_CFC_ (* Continuous Function Chart, elements in execution order *)
#0 SHU6_P2_M_MAXSPEED <= SHU6_P2_M_MAXSPEED_CH
#1 <>(SHU6_P2_M_MAXSPEED_CH, SHU6_P2_M_MAXSPEED_CH_OLD)
#2 RS_RUCH:RS(SET: #1, RESET1: #4.Q)
#3 V_RUCH <= #2.Q1
#4 TON_RUCH:TON(IN: #2.Q1, PT: T#10s)
#5 AND(SHU6_P2_YA3_M_UST_VKL_UVEL_CHAST, SHU6_P2_YA4_M_UST_VKL_UVEL_CHAST, SHU6_P2_UST_RE_RABOTA)
#6 TON_STER_1:TON(IN: #5, PT: T#60s)
#7 OR(#6.Q, SHU6_P2_M_SB2_STER_REG)
#8 AND(#7, SHU6_P2_UST_RE_RABOTA, NOT V_RUCH)
#9 OR(V_RUCH, SHU6_P2_UST_RE_PUSK)
#10 SEL(#8, SHU6_P2_SPEEDMOTOR, SHU6_P2_M_MAXSPEED)
#11 AND(#8, NOT V_RUCH)
#12 SEL(#11, SHU6_P2_M_USKORENIE_PUSK, SHU6_P2_M_USKORENIE_UPR)
#13 OR(SHU6_P2_YA3_B_UST_VKL_STER_REG, SHU6_P2_YA4_B_UST_VKL_STER_REG)
#14 AND(SHU6_P2_UST_RE_RABOTA, #13)
#15 TON_STER_2:TON(IN: #14, PT: T#60s)
#16 AND(NOT SHU6_P2_M_SB2_STER_REG, #15.Q, SHU6_P2_UST_RE_RABOTA, NOT V_RUCH)
#17 SEL(#16, #10, SHU6_P2_M_MINSPEED)
#18 SEL(#9, #17, SHU6_P2_M_MAXSPEED)
#19 SEL(SHU6_P2_UST_SOST_VKL, 0, #18)
#20 AND(#16, NOT V_RUCH)
#21 SEL(#20, SHU6_P2_M_ZAMEDLENIE_OST, SHU6_P2_M_ZAMEDLENIE_UPR)
#22 SEL(SHU6_P2_UST_SET_STOP, #21, 1000)
#23 RR:RAMP_REAL(#19, #12, #22, T#1s, -)
#24 SHU6_P2_SPEEDMOTOR <= #23
#25 MOVE(EN: SHU6_P2_SA1_DO1, #23)
#26 SEL(#25.ENO, 0, #25)
#27 SEL(SHU6_P2_SA1_DI2_M, #26, SHU6_P2_M_ZAD_RUCH)
#28 SHU6_P2_ZAD_VN <= #27
#29 MOVE(EN: SHU6_V2_SA3_DO3, #23)
#30 SEL(#29.ENO, 0, #29)
#31 SEL(SHU6_V2_SA2_DI6_M, #30, SHU6_V2_M_ZAD_RUCH)
#32 SHU6_V2_ZAD_VN <= #31
#33 SHU6_P2_M_MAXSPEED_CH_OLD <= SHU6_P2_M_MAXSPEED_CH
#34 RT_KOMVKL_2:R_TRIG(CLK: TRUE)
#35 MOVE(EN: #34.Q, 5)
#36 SHU6_P2_M_ZAD_RUCH <= #35
_END_CFC_
END_PROGRAM

(* POU IM/MP2/MP2_1, CFC *)
PROGRAM MP2_1
VAR
	RS_M1: RS;

	startDelay_M1: TIME := T#0s;
	stopDelay_M1: TIME := T#0s;
	delayFBC_M1: TIME := T#30S;
	feedbPT_M1: TIME := T#120s;
	delayFBP_M1: TIME := T#30s;

	fb_HVACMS_M1: FB_HVACMotor1Speed;
	fb_HVACPIDC_M1: FB_HVACPIDCtrl;

	deadRange: REAL := 0.1;
	rKp: REAL := 1;
	tTi: TIME;
	tTv: TIME := T#0s;
	tTd: TIME := T#0s;
	direction: BOOL;
	rYMin: REAL;
	Dint_Ti: DINT;
	set: BOOL;
	reset: BOOL;
	resetContr: BOOL;
	SR_VKL: SR;
	TON_PUSK: TON;
	RT_PUSK: R_TRIG;
	TON_NP2_OTKAZ: TON;
END_VAR
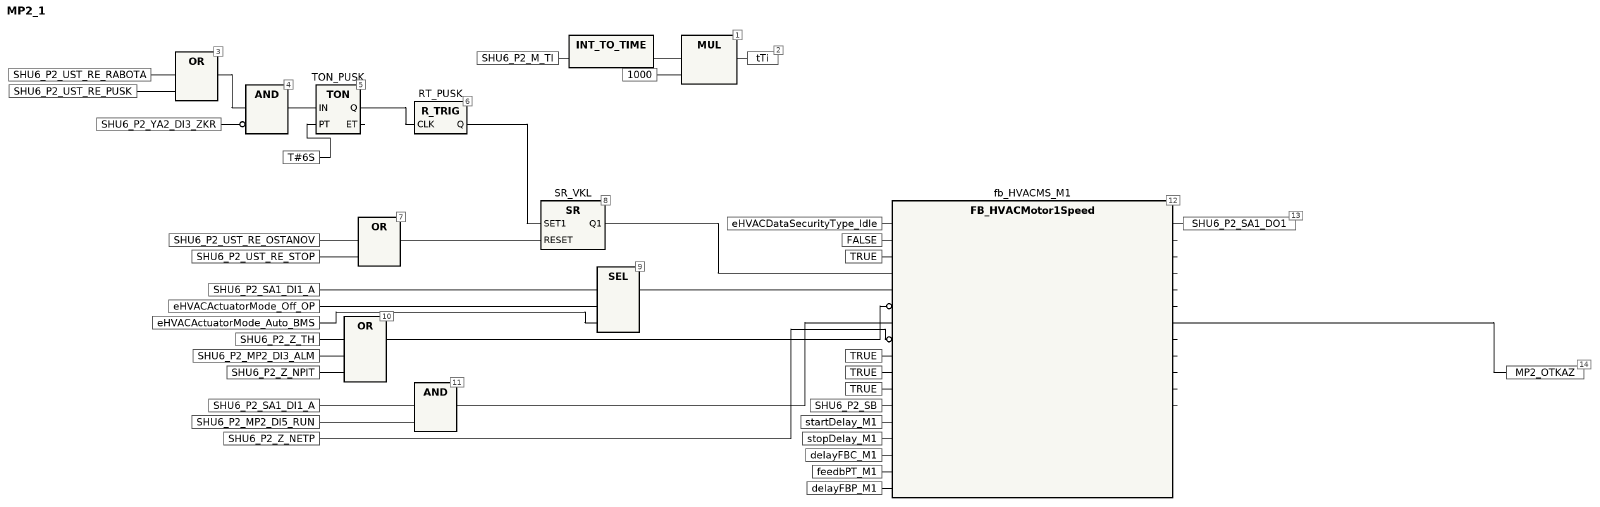
_CFC_ (* Continuous Function Chart, elements in execution order *)
#0 INT_TO_TIME(SHU6_P2_M_TI)
#1 MUL(#0, 1000)
#2 tTi <= #1
#3 OR(SHU6_P2_UST_RE_RABOTA, SHU6_P2_UST_RE_PUSK)
#4 AND(#3, NOT SHU6_P2_YA2_DI3_ZKR)
#5 TON_PUSK:TON(IN: #4, PT: T#6S)
#6 RT_PUSK:R_TRIG(CLK: #5.Q)
#7 OR(SHU6_P2_UST_RE_OSTANOV, SHU6_P2_UST_RE_STOP)
#8 SR_VKL:SR(SET1: #6.Q, RESET: #7)
#9 SEL(SHU6_P2_SA1_DI1_A, eHVACActuatorMode_Off_OP, eHVACActuatorMode_Auto_BMS)
#10 OR(SHU6_P2_Z_TH, SHU6_P2_MP2_DI3_ALM, SHU6_P2_Z_NPIT)
#11 AND(SHU6_P2_SA1_DI1_A, SHU6_P2_MP2_DI5_RUN)
#12 fb_HVACMS_M1:FB_HVACMotor1Speed(eHVACDataSecurityType_Idle, FALSE, TRUE, #8.Q1, #9, NOT #10, #11, NOT SHU6_P2_Z_NETP, TRUE, TRUE, TRUE, SHU6_P2_SB, startDelay_M1, stopDelay_M1, delayFBC_M1, feedbPT_M1, delayFBP_M1)
#13 SHU6_P2_SA1_DO1 <= #12.out 1
#14 MP2_OTKAZ <= #12.out 7
_END_CFC_
END_PROGRAM

(* POU IM/P1_Upr, CFC *)
PROGRAM P1_Upr
VAR
	fb_HVACMS_P1: FB_HVACMotor1Speed;
	SR_P1: SR;
	startDelay_P1: TIME := T#0s;
	stopDelay_P1: TIME := T#0s;
	delayFBC_P1: TIME;
	feedbPT_P1: TIME :=T#10s ;
	delayFBP_P1: TIME := T#10s;
	TON_P1_OTKL_Leto: TON;
	TON_P1_VKL_Leto: TON;
END_VAR
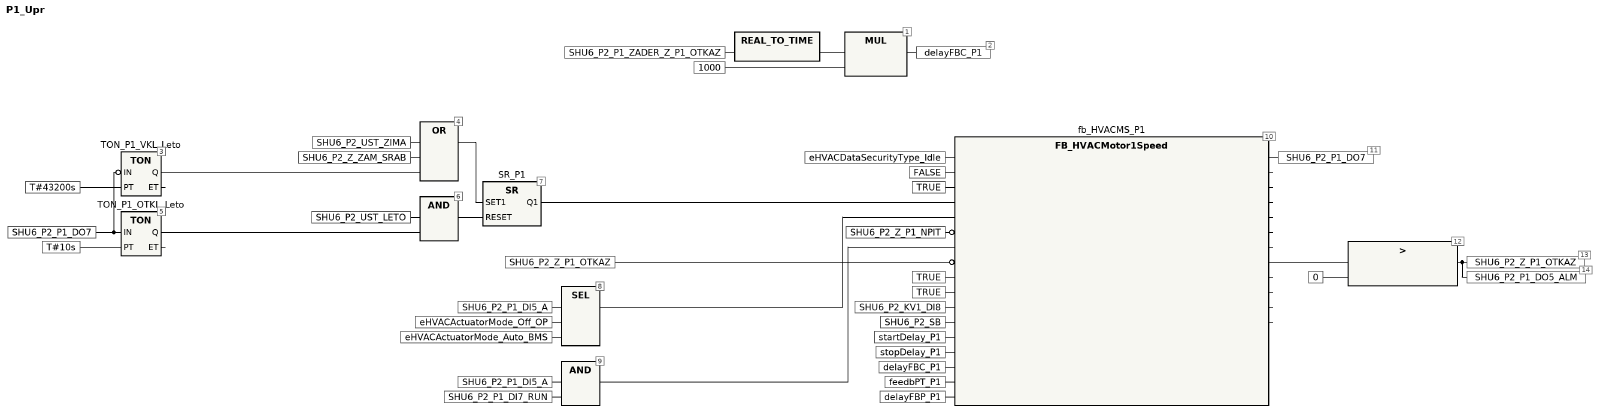
